// TIA Portal project "Sistema_de_silos" (V16)

(* hardware
DEVICE "S7-1200 station_1"  S7-1200 Station
   slot 0: "Rack_0"  S7-1200 Rack  Rack  V1.0
   slot 1: "PLC_1"  CPU 1215C DC/DC/Rly  6ES7 215-1HG40-0XB0  V4.4
*)

// ===== PLC "PLC_1"  CPU 1215C DC/DC/Rly =====

VAR_GLOBAL   // PLC tag table "Inputs"
   "bt0" AT %I0.0 : Bool;   // botao automático
   "bt1" AT %I0.1 : Bool;   // botao manual
   "bt2" AT %I0.2 : Bool;   // botao reset
   "bt3" AT %I0.3 : Bool;   // botao Emg
   "b01" AT %I0.4 : Bool;   // sensor B01 Silo 1 Nivel Minimo
   "b02" AT %I0.5 : Bool;   // sensor B02 Silo 1 Nivel Maximo
   "b03" AT %I0.6 : Bool;   // sensor B03 Damper aberto silo 2
   "b04" AT %I0.7 : Bool;   // sensor B04 Damper aberto silo 3
   "b05" AT %I1.0 : Bool;   // sensor B05 Silo 2 Nivel Minimo
   "b06" AT %I1.1 : Bool;   // sensor B06 Silo 2 Nivel Máximo
   "b07" AT %I1.2 : Bool;   // sensor B07 Silo 3 Nivel Minimo
   "b08" AT %I1.3 : Bool;   // sensor B08 Silo 3 Nivel Máximo
   "b09" AT %I1.4 : Bool;   // sensor B09 Damper Fechado
   "Reserva" AT %I1.5 : Bool;   // sensor B10 Valvula Silo 2 Fechada
END_VAR

VAR_GLOBAL   // PLC tag table "Outputs"
   "x0.0" AT %Q0.0 : Bool;   // sinalizacao verde
   "x0.1" AT %Q0.1 : Bool;   // sinalizacao amarelo
   "x0.2" AT %Q0.2 : Bool;   // sinalizacao vermelho
   "k0.3" AT %Q0.3 : Bool;   // damper silo 2
   "k0.4" AT %Q0.4 : Bool;   // damper fecha
   "k0.5" AT %Q0.5 : Bool;   // Liga Transportador Silo 2
   "k0.6" AT %Q0.6 : Bool;   // Liga Transportador Silo 3
   "k0.7" AT %Q0.7 : Bool;   // Abre Valvula Silo 1
   "k10" AT %Q1.0 : Bool;   // Abre Valvula Silo 2
   "k11" AT %Q1.1 : Bool;   // damper silo 3
END_VAR

VAR_GLOBAL   // PLC tag table "Memories"
   "Memoria_Auxiliar_Erro_Silo" AT %M0.1 : Bool;
   "ST_FALHA" AT %M0.2 : Bool;
END_VAR

DATA_BLOCK "DB_Geral"   // DB1
{ S7_Optimized_Access := 'TRUE' }
VERSION : 0.1
   VAR
      automatico : Bool;   // Estado automatico
      manual : Bool;   // Estado Manual
      Emg : Bool;   // Estado Emergência
      Falha : Struct   // Estado Falha
         Falha_Desabastecimento_Silo2 : Bool;
         Falha_Desabastecimento_Silo3 : Bool;
         Falha_Desabastecimento_SiloPrincipal : Bool;
         Falha_Sensores_Silo2 : Bool;
         Falha_Sensores_Silo3 : Bool;
         Falha_Sensores_SiloPrincipal : Bool;
      END_STRUCT;
      Diametro_Valvula : Real := 0.1;
      Volume_sensor : Int := 3;
      Volume_maximo_minimo : Int := 7;
      Time_Dint_Valvula : DInt;
      Time_Dint_TempoErro : DInt;
      Time_Valvula : Time;
      Time_TempoErro : Time;
      Sequencia : Struct   // Sequencia Operacional
         Acao : Array[0..50] of Bool;
         Passos : Int;
      END_STRUCT;
      "Status Silo Principal" : Struct   // Status do Silo Principal
         Maximo : Bool;
         Minimo : Bool;
         Desabastecido : Bool;
         Posicao_Produto : Int;
      END_STRUCT;
      "Status Silo 2" : Struct   // Status do Silo 2
         Maximo : Bool;
         Minimo : Bool;
         Desabastecido : Bool;
         Posicao_Produto : Int;
      END_STRUCT;
      "Status Silo 3" : Struct   // Status do Silo 3
         Maximo : Bool;
         Minimo : Bool;
         Desabastecido : Bool;
         Posicao_Produto : Bool;
      END_STRUCT;
      "Status Transportador" : Struct   // Status Transportadores
         "Transportador 1" : Bool;
         "Transportador 2" : Bool;
      END_STRUCT;
      "Status Damper" : Struct   // Status do Damper
         Ligado : Bool;
         "Silo 2" : Bool;
         "Silo 3" : Bool;
      END_STRUCT;
      "Status Valvulas" : Struct   // Status das Valvulas
         "Valvula Silo 2" : Bool;
         "Valvula Silo 3" : Bool;
      END_STRUCT;
   END_VAR
BEGIN
   // Sequencia.Acao[20] : Ação 20
   // Sequencia.Acao[30] : Ação 30
   // Sequencia.Acao[31] : Ação 31
   // Sequencia.Acao[21] : Ação 21
   // Sequencia.Acao[22] : Ação 22
   // Sequencia.Acao[40] : Ação 40
   // Sequencia.Acao[41] : Ação 41
   // Sequencia.Acao[10] : Ação 10
   // Sequencia.Acao[11] : Ação 11
END_DATA_BLOCK

DATA_BLOCK "DB_Inputs"   // DB2
{ S7_Optimized_Access := 'TRUE' }
VERSION : 0.1
   VAR
      bt0 : Bool;   // botao automático
      bt1 : Bool;   // botao manual
      bt2 : Bool;   // botao reset
      bt3 : Bool;   // botao Emg
      bt4 : Bool;   // botao Abre Valvula 2
      bt5 : Bool;   // botao Abre Valvula 3
      b01 : Bool;   // sensor B01 Silo 1 Nivel Minimo
      b02 : Bool;   // sensor B02 Silo 1 Nivel Maximo
      b03 : Bool;   // sensor B03 Damper aberto silo 2
      b04 : Bool;   // sensor B04 Damper aberto silo 3
      b05 : Bool;   // sensor B05 Silo 2 Nivel Minimo
      b06 : Bool;   // sensor B06 Silo 2 Nivel Máximo
      b07 : Bool;   // sensor B07 Silo 3 Nivel Minimo
      b08 : Bool;   // sensor B08 Silo 3 Nivel Máximo
      b09 : Bool;   // sensor B09 Damper Fechado
   END_VAR
BEGIN
END_DATA_BLOCK

DATA_BLOCK "DB_Outputs"   // DB3
{ S7_Optimized_Access := 'TRUE' }
VERSION : 0.1
   VAR
      "x0.0" : Bool;   // sinalizacao verde
      "x0.1" : Bool;   // sinalizacao amarelo
      "x0.2" : Bool;   // sinalizacao vermelho
      "k0.3" : Bool;   // damper Abre silo 2
      "k0.4" : Bool;   // damper Abre silo 3
      "k0.5" : Bool;   // Liga Transportador Silo 2
      "k0.6" : Bool;   // Liga Transportador Silo 3
      "k0.7" : Bool;   // Abre Valvula Silo 2
      k10 : Bool;   // Abre Valvula Silo 3
      k11 : Bool;   // Abastece Silo Principal
   END_VAR
BEGIN
END_DATA_BLOCK

// folder: System blocks/Program resources

DATA_BLOCK "IEC_Timer_0_DB_TOF_VALVULA2"   // DB4
{ S7_Optimized_Access := 'TRUE' }
AUTHOR : Simatic
FAMILY : IEC
NAME : IEC_TMR
VERSION : 1.0
// stored: InstanceOfName IEC_TIMER
"IEC_TIMER"
BEGIN
END_DATA_BLOCK

DATA_BLOCK "IEC_Timer_0_DB_TON_TempoErro"   // DB5
{ S7_Optimized_Access := 'TRUE' }
AUTHOR : Simatic
FAMILY : IEC
NAME : IEC_TMR
VERSION : 1.0
// stored: InstanceOfName IEC_TIMER
"IEC_TIMER"
BEGIN
END_DATA_BLOCK

// folder: (top level)

FUNCTION "FC_Geral" : Void   // FC1, LAD
{ S7_Optimized_Access := 'TRUE' }
VERSION : 0.1
   VAR_TEMP   // added for the SCL form of the ladder/FBD networks
      _w1 : Bool;
   END_VAR
BEGIN

REGION Network 1: Estado Emergencia
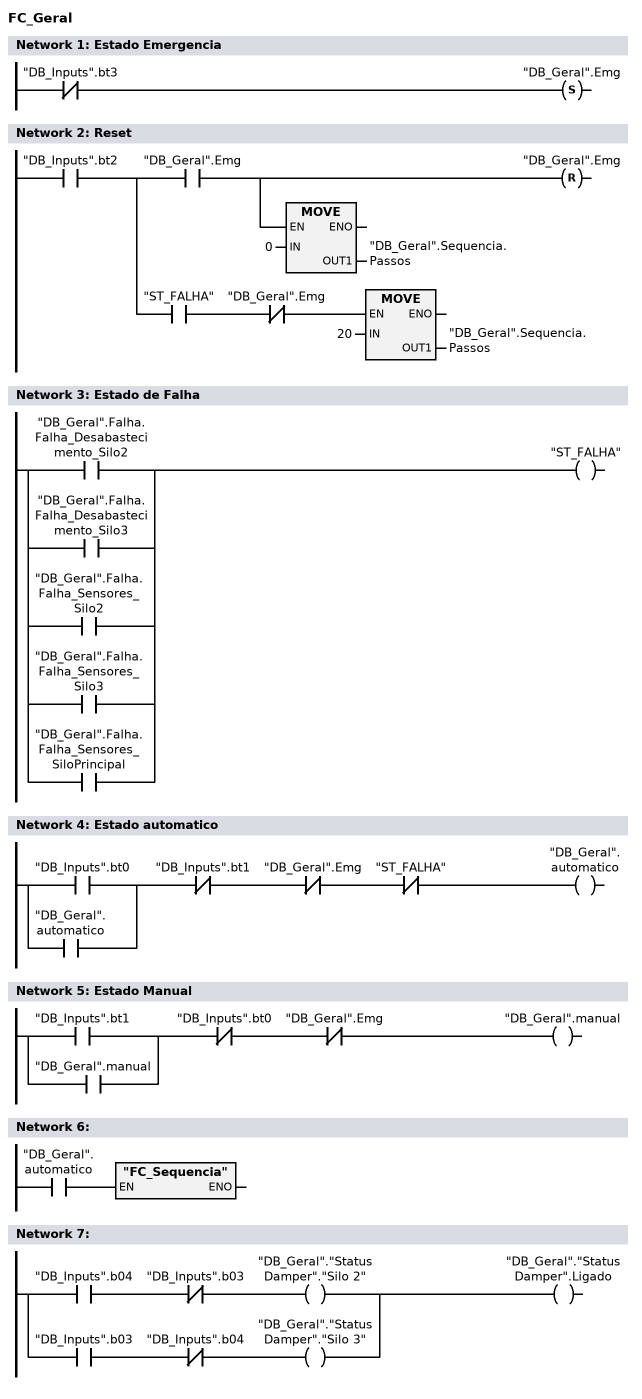
   RUNG wire#powerrail
      I_Contact( "DB_Inputs".bt3 )
      S_Coil( "DB_Geral".Emg )
   END_RUNG
   // the same network as SCL:
   IF NOT "DB_Inputs".bt3 THEN "DB_Geral".Emg := TRUE; END_IF;
END_REGION

REGION Network 2: Reset
   RUNG wire#powerrail
      Contact( "DB_Inputs".bt2 )
      wire#w1
      Contact( "DB_Geral".Emg )
      wire#w2
      R_Coil( "DB_Geral".Emg )
   END_RUNG
   RUNG wire#w2
      Move(in := 0, out1 => "DB_Geral".Sequencia.Passos)
   END_RUNG
   RUNG wire#w1
      Contact( "ST_FALHA" )
      I_Contact( "DB_Geral".Emg )
      Move(in := 20, out1 => "DB_Geral".Sequencia.Passos)
   END_RUNG
   // the same network as SCL:
   #_w1 := "DB_Inputs".bt2 AND "DB_Geral".Emg;
   IF #_w1 THEN
       "DB_Geral".Emg := FALSE;
       "DB_Geral".Sequencia.Passos := 0;
   END_IF;
   IF "DB_Inputs".bt2 AND "ST_FALHA" AND NOT "DB_Geral".Emg THEN "DB_Geral".Sequencia.Passos := 20; END_IF;
END_REGION

REGION Network 3: Estado de Falha
   RUNG wire#powerrail
      Contact( "DB_Geral".Falha.Falha_Desabastecimento_Silo2 )
      wire#w1
      Coil( "ST_FALHA" )
   END_RUNG
   RUNG wire#powerrail
      Contact( "DB_Geral".Falha.Falha_Desabastecimento_Silo3 )
   END_RUNG wire#w1
   RUNG wire#powerrail
      Contact( "DB_Geral".Falha.Falha_Sensores_Silo2 )
   END_RUNG wire#w1
   RUNG wire#powerrail
      Contact( "DB_Geral".Falha.Falha_Sensores_Silo3 )
   END_RUNG wire#w1
   RUNG wire#powerrail
      Contact( "DB_Geral".Falha.Falha_Sensores_SiloPrincipal )
   END_RUNG wire#w1
   // the same network as SCL:
   "ST_FALHA" := "DB_Geral".Falha.Falha_Desabastecimento_Silo2 OR "DB_Geral".Falha.Falha_Desabastecimento_Silo3 OR "DB_Geral".Falha.Falha_Sensores_Silo2 OR "DB_Geral".Falha.Falha_Sensores_Silo3 OR "DB_Geral".Falha.Falha_Sensores_SiloPrincipal;
END_REGION

REGION Network 4: Estado automatico
   RUNG wire#powerrail
      Contact( "DB_Inputs".bt0 )
      wire#w1
      I_Contact( "DB_Inputs".bt1 )
      I_Contact( "DB_Geral".Emg )
      I_Contact( "ST_FALHA" )
      Coil( "DB_Geral".automatico )
   END_RUNG
   RUNG wire#powerrail
      Contact( "DB_Geral".automatico )
   END_RUNG wire#w1
   // the same network as SCL:
   "DB_Geral".automatico := ("DB_Inputs".bt0 OR "DB_Geral".automatico) AND NOT "DB_Inputs".bt1 AND NOT "DB_Geral".Emg AND NOT "ST_FALHA";
END_REGION

REGION Network 5: Estado Manual
   RUNG wire#powerrail
      Contact( "DB_Inputs".bt1 )
      wire#w1
      I_Contact( "DB_Inputs".bt0 )
      I_Contact( "DB_Geral".Emg )
      Coil( "DB_Geral".manual )
   END_RUNG
   RUNG wire#powerrail
      Contact( "DB_Geral".manual )
   END_RUNG wire#w1
   // the same network as SCL:
   "DB_Geral".manual := ("DB_Inputs".bt1 OR "DB_Geral".manual) AND NOT "DB_Inputs".bt0 AND NOT "DB_Geral".Emg;
END_REGION

REGION Network 6
   RUNG wire#powerrail
      Contact( "DB_Geral".automatico )
      "FC_Sequencia"()
   END_RUNG
   // the same network as SCL:
   IF "DB_Geral".automatico THEN "FC_Sequencia"(); END_IF;
END_REGION

REGION Network 7
   RUNG wire#powerrail
      Contact( "DB_Inputs".b04 )
      I_Contact( "DB_Inputs".b03 )
      Coil( "DB_Geral"."Status Damper"."Silo 2" )
      wire#w1
      Coil( "DB_Geral"."Status Damper".Ligado )
   END_RUNG
   RUNG wire#powerrail
      Contact( "DB_Inputs".b03 )
      I_Contact( "DB_Inputs".b04 )
      Coil( "DB_Geral"."Status Damper"."Silo 3" )
   END_RUNG wire#w1
   // the same network as SCL:
   "DB_Geral"."Status Damper"."Silo 2" := "DB_Inputs".b04 AND NOT "DB_Inputs".b03;
   "DB_Geral"."Status Damper"."Silo 3" := "DB_Inputs".b03 AND NOT "DB_Inputs".b04;
   "DB_Geral"."Status Damper".Ligado := "DB_Geral"."Status Damper"."Silo 2" OR "DB_Geral"."Status Damper"."Silo 3";
END_REGION
END_FUNCTION

FUNCTION "FC_Espelho_Outputs" : Void   // FC2, LAD
{ S7_Optimized_Access := 'TRUE' }
VERSION : 0.1
BEGIN

REGION Network 1: sinalizacao verde
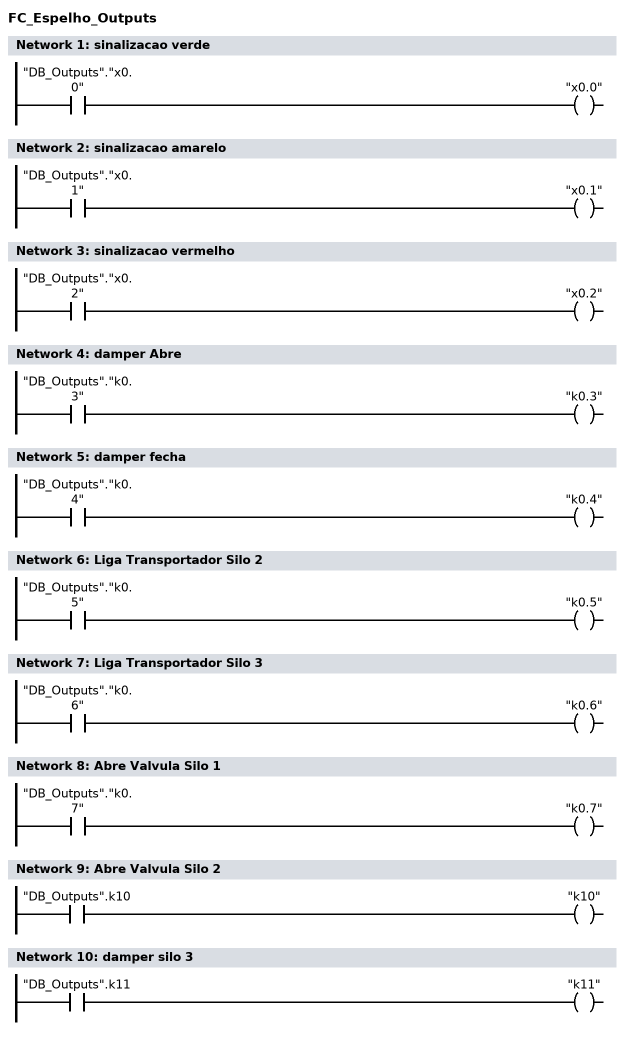
   RUNG wire#powerrail
      Contact( "DB_Outputs"."x0.0" )
      Coil( "x0.0" )
   END_RUNG
   // the same network as SCL:
   "x0.0" := "DB_Outputs"."x0.0";
END_REGION

REGION Network 2: sinalizacao amarelo
   RUNG wire#powerrail
      Contact( "DB_Outputs"."x0.1" )
      Coil( "x0.1" )
   END_RUNG
   // the same network as SCL:
   "x0.1" := "DB_Outputs"."x0.1";
END_REGION

REGION Network 3: sinalizacao vermelho
   RUNG wire#powerrail
      Contact( "DB_Outputs"."x0.2" )
      Coil( "x0.2" )
   END_RUNG
   // the same network as SCL:
   "x0.2" := "DB_Outputs"."x0.2";
END_REGION

REGION Network 4: damper Abre
   RUNG wire#powerrail
      Contact( "DB_Outputs"."k0.3" )
      Coil( "k0.3" )
   END_RUNG
   // the same network as SCL:
   "k0.3" := "DB_Outputs"."k0.3";
END_REGION

REGION Network 5: damper fecha
   RUNG wire#powerrail
      Contact( "DB_Outputs"."k0.4" )
      Coil( "k0.4" )
   END_RUNG
   // the same network as SCL:
   "k0.4" := "DB_Outputs"."k0.4";
END_REGION

REGION Network 6: Liga Transportador Silo 2
   RUNG wire#powerrail
      Contact( "DB_Outputs"."k0.5" )
      Coil( "k0.5" )
   END_RUNG
   // the same network as SCL:
   "k0.5" := "DB_Outputs"."k0.5";
END_REGION

REGION Network 7: Liga Transportador Silo 3
   RUNG wire#powerrail
      Contact( "DB_Outputs"."k0.6" )
      Coil( "k0.6" )
   END_RUNG
   // the same network as SCL:
   "k0.6" := "DB_Outputs"."k0.6";
END_REGION

REGION Network 8: Abre Valvula Silo 1
   RUNG wire#powerrail
      Contact( "DB_Outputs"."k0.7" )
      Coil( "k0.7" )
   END_RUNG
   // the same network as SCL:
   "k0.7" := "DB_Outputs"."k0.7";
END_REGION

REGION Network 9: Abre Valvula Silo 2
   RUNG wire#powerrail
      Contact( "DB_Outputs".k10 )
      Coil( "k10" )
   END_RUNG
   // the same network as SCL:
   "k10" := "DB_Outputs".k10;
END_REGION

REGION Network 10: damper silo 3
   RUNG wire#powerrail
      Contact( "DB_Outputs".k11 )
      Coil( "k11" )
   END_RUNG
   // the same network as SCL:
   "k11" := "DB_Outputs".k11;
END_REGION
END_FUNCTION

FUNCTION "FC_Espelho_Inputs" : Void   // FC3, LAD
{ S7_Optimized_Access := 'TRUE' }
VERSION : 0.1
BEGIN

REGION Network 1: botao automático
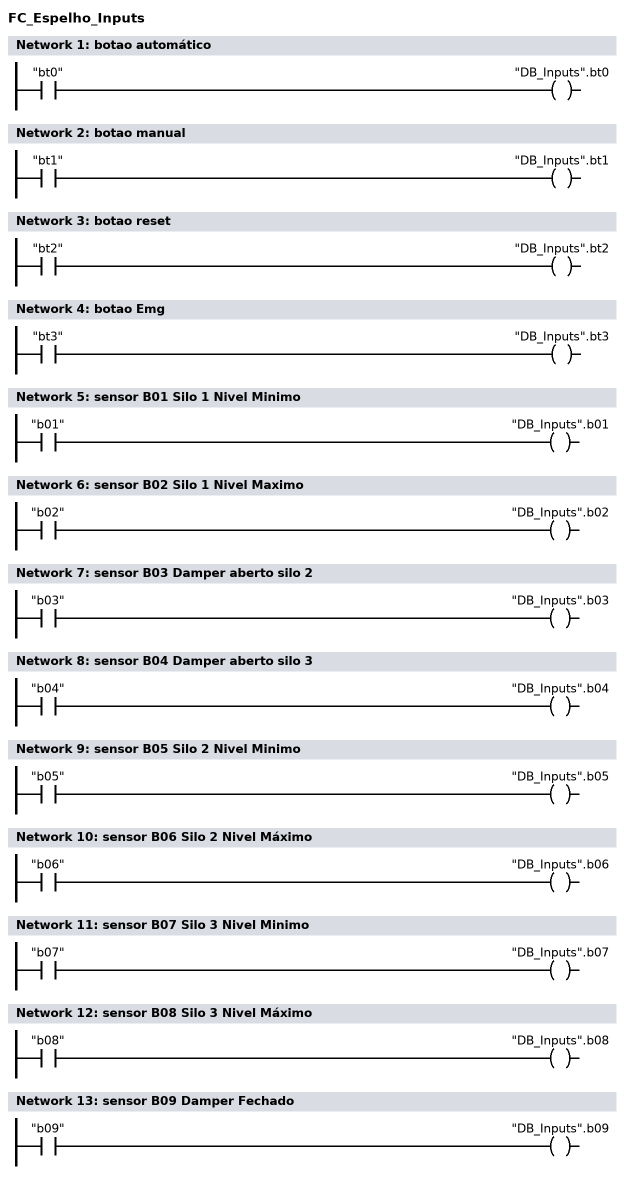
   RUNG wire#powerrail
      Contact( "bt0" )
      Coil( "DB_Inputs".bt0 )
   END_RUNG
   // the same network as SCL:
   "DB_Inputs".bt0 := "bt0";
END_REGION

REGION Network 2: botao manual
   RUNG wire#powerrail
      Contact( "bt1" )
      Coil( "DB_Inputs".bt1 )
   END_RUNG
   // the same network as SCL:
   "DB_Inputs".bt1 := "bt1";
END_REGION

REGION Network 3: botao reset
   RUNG wire#powerrail
      Contact( "bt2" )
      Coil( "DB_Inputs".bt2 )
   END_RUNG
   // the same network as SCL:
   "DB_Inputs".bt2 := "bt2";
END_REGION

REGION Network 4: botao Emg
   RUNG wire#powerrail
      Contact( "bt3" )
      Coil( "DB_Inputs".bt3 )
   END_RUNG
   // the same network as SCL:
   "DB_Inputs".bt3 := "bt3";
END_REGION

REGION Network 5: sensor B01 Silo 1 Nivel Minimo
   RUNG wire#powerrail
      Contact( "b01" )
      Coil( "DB_Inputs".b01 )
   END_RUNG
   // the same network as SCL:
   "DB_Inputs".b01 := "b01";
END_REGION

REGION Network 6: sensor B02 Silo 1 Nivel Maximo
   RUNG wire#powerrail
      Contact( "b02" )
      Coil( "DB_Inputs".b02 )
   END_RUNG
   // the same network as SCL:
   "DB_Inputs".b02 := "b02";
END_REGION

REGION Network 7: sensor B03 Damper aberto silo 2
   RUNG wire#powerrail
      Contact( "b03" )
      Coil( "DB_Inputs".b03 )
   END_RUNG
   // the same network as SCL:
   "DB_Inputs".b03 := "b03";
END_REGION

REGION Network 8: sensor B04 Damper aberto silo 3
   RUNG wire#powerrail
      Contact( "b04" )
      Coil( "DB_Inputs".b04 )
   END_RUNG
   // the same network as SCL:
   "DB_Inputs".b04 := "b04";
END_REGION

REGION Network 9: sensor B05 Silo 2 Nivel Minimo
   RUNG wire#powerrail
      Contact( "b05" )
      Coil( "DB_Inputs".b05 )
   END_RUNG
   // the same network as SCL:
   "DB_Inputs".b05 := "b05";
END_REGION

REGION Network 10: sensor B06 Silo 2 Nivel Máximo
   RUNG wire#powerrail
      Contact( "b06" )
      Coil( "DB_Inputs".b06 )
   END_RUNG
   // the same network as SCL:
   "DB_Inputs".b06 := "b06";
END_REGION

REGION Network 11: sensor B07 Silo 3 Nivel Minimo
   RUNG wire#powerrail
      Contact( "b07" )
      Coil( "DB_Inputs".b07 )
   END_RUNG
   // the same network as SCL:
   "DB_Inputs".b07 := "b07";
END_REGION

REGION Network 12: sensor B08 Silo 3 Nivel Máximo
   RUNG wire#powerrail
      Contact( "b08" )
      Coil( "DB_Inputs".b08 )
   END_RUNG
   // the same network as SCL:
   "DB_Inputs".b08 := "b08";
END_REGION

REGION Network 13: sensor B09 Damper Fechado
   RUNG wire#powerrail
      Contact( "b09" )
      Coil( "DB_Inputs".b09 )
   END_RUNG
   // the same network as SCL:
   "DB_Inputs".b09 := "b09";
END_REGION
END_FUNCTION

FUNCTION "FC_Sequencia" : Void   // FC4, LAD
{ S7_Optimized_Access := 'TRUE' }
VERSION : 0.1
   VAR_TEMP   // added for the SCL form of the ladder/FBD networks
      _w1 : Bool;
   END_VAR
BEGIN

REGION Network 1
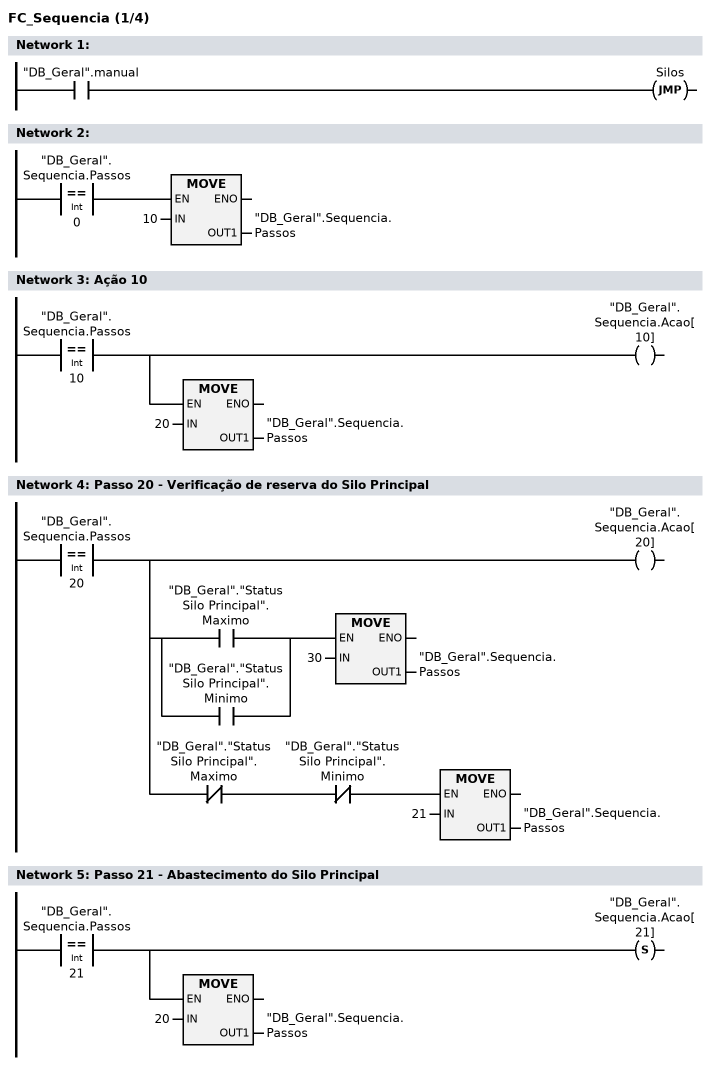
   RUNG wire#powerrail
      Contact( "DB_Geral".manual )
      JumpCoil( Silos )
   END_RUNG
   // the same network as SCL:
   IF "DB_Geral".manual THEN GOTO Silos; END_IF;
END_REGION

REGION Network 2
   RUNG wire#powerrail
      { S7_Templates := "SrcType := Int" } EQ_Contact(in1 := "DB_Geral".Sequencia.Passos, in2 := 0)
      Move(in := 10, out1 => "DB_Geral".Sequencia.Passos)
   END_RUNG
   // the same network as SCL:
   IF "DB_Geral".Sequencia.Passos = 0 THEN "DB_Geral".Sequencia.Passos := 10; END_IF;
END_REGION

REGION Network 3: Ação 10
   RUNG wire#powerrail
      { S7_Templates := "SrcType := Int" } EQ_Contact(in1 := "DB_Geral".Sequencia.Passos, in2 := 10)
      wire#w1
      Coil( "DB_Geral".Sequencia.Acao[10] )
   END_RUNG
   RUNG wire#w1
      Move(in := 20, out1 => "DB_Geral".Sequencia.Passos)
   END_RUNG
   // the same network as SCL:
   "DB_Geral".Sequencia.Acao[10] := "DB_Geral".Sequencia.Passos = 10;
   IF "DB_Geral".Sequencia.Passos = 10 THEN "DB_Geral".Sequencia.Passos := 20; END_IF;
END_REGION

REGION Network 4: Passo 20 - Verificação de reserva do Silo Principal
   RUNG wire#powerrail
      { S7_Templates := "SrcType := Int" } EQ_Contact(in1 := "DB_Geral".Sequencia.Passos, in2 := 20)
      wire#w1
      Coil( "DB_Geral".Sequencia.Acao[20] )
   END_RUNG
   RUNG wire#w1
      Contact( "DB_Geral"."Status Silo Principal".Maximo )
      wire#w2
      Move(in := 30, out1 => "DB_Geral".Sequencia.Passos)
   END_RUNG
   RUNG wire#w1
      Contact( "DB_Geral"."Status Silo Principal".Minimo )
   END_RUNG wire#w2
   RUNG wire#w1
      I_Contact( "DB_Geral"."Status Silo Principal".Maximo )
      I_Contact( "DB_Geral"."Status Silo Principal".Minimo )
      Move(in := 21, out1 => "DB_Geral".Sequencia.Passos)
   END_RUNG
   // the same network as SCL:
   "DB_Geral".Sequencia.Acao[20] := "DB_Geral".Sequencia.Passos = 20;
   #_w1 := "DB_Geral".Sequencia.Passos = 20;
   IF ("DB_Geral".Sequencia.Passos = 20) AND ("DB_Geral"."Status Silo Principal".Maximo OR "DB_Geral"."Status Silo Principal".Minimo) THEN
       "DB_Geral".Sequencia.Passos := 30;
   END_IF;
   IF #_w1 AND NOT "DB_Geral"."Status Silo Principal".Maximo AND NOT "DB_Geral"."Status Silo Principal".Minimo THEN
       "DB_Geral".Sequencia.Passos := 21;
   END_IF;
END_REGION

REGION Network 5: Passo 21 - Abastecimento do Silo Principal
   RUNG wire#powerrail
      { S7_Templates := "SrcType := Int" } EQ_Contact(in1 := "DB_Geral".Sequencia.Passos, in2 := 21)
      wire#w1
      S_Coil( "DB_Geral".Sequencia.Acao[21] )
   END_RUNG
   RUNG wire#w1
      Move(in := 20, out1 => "DB_Geral".Sequencia.Passos)
   END_RUNG
   // the same network as SCL:
   IF "DB_Geral".Sequencia.Passos = 21 THEN
       "DB_Geral".Sequencia.Acao[21] := TRUE;
       "DB_Geral".Sequencia.Passos := 20;
   END_IF;
END_REGION

REGION Network 6: Passo 30 - Verificação do Silo 2
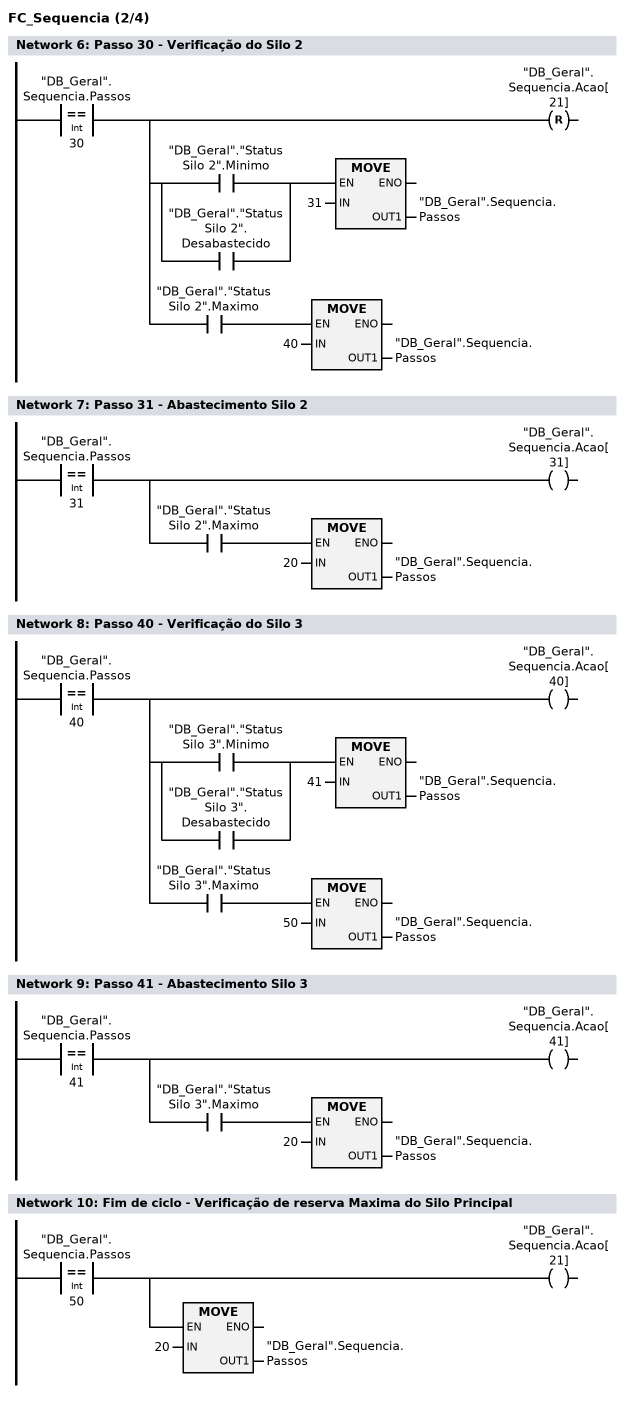
   RUNG wire#powerrail
      { S7_Templates := "SrcType := Int" } EQ_Contact(in1 := "DB_Geral".Sequencia.Passos, in2 := 30)
      wire#w1
      R_Coil( "DB_Geral".Sequencia.Acao[21] )
   END_RUNG
   RUNG wire#w1
      Contact( "DB_Geral"."Status Silo 2".Minimo )
      wire#w2
      Move(in := 31, out1 => "DB_Geral".Sequencia.Passos)
   END_RUNG
   RUNG wire#w1
      Contact( "DB_Geral"."Status Silo 2".Desabastecido )
   END_RUNG wire#w2
   RUNG wire#w1
      Contact( "DB_Geral"."Status Silo 2".Maximo )
      Move(in := 40, out1 => "DB_Geral".Sequencia.Passos)
   END_RUNG
   // the same network as SCL:
   #_w1 := "DB_Geral".Sequencia.Passos = 30;
   IF #_w1 THEN "DB_Geral".Sequencia.Acao[21] := FALSE; END_IF;
   IF #_w1 AND ("DB_Geral"."Status Silo 2".Minimo OR "DB_Geral"."Status Silo 2".Desabastecido) THEN
       "DB_Geral".Sequencia.Passos := 31;
   END_IF;
   IF #_w1 AND "DB_Geral"."Status Silo 2".Maximo THEN "DB_Geral".Sequencia.Passos := 40; END_IF;
END_REGION

REGION Network 7: Passo 31 - Abastecimento Silo 2
   RUNG wire#powerrail
      { S7_Templates := "SrcType := Int" } EQ_Contact(in1 := "DB_Geral".Sequencia.Passos, in2 := 31)
      wire#w1
      Coil( "DB_Geral".Sequencia.Acao[31] )
   END_RUNG
   RUNG wire#w1
      Contact( "DB_Geral"."Status Silo 2".Maximo )
      Move(in := 20, out1 => "DB_Geral".Sequencia.Passos)
   END_RUNG
   // the same network as SCL:
   "DB_Geral".Sequencia.Acao[31] := "DB_Geral".Sequencia.Passos = 31;
   IF ("DB_Geral".Sequencia.Passos = 31) AND "DB_Geral"."Status Silo 2".Maximo THEN
       "DB_Geral".Sequencia.Passos := 20;
   END_IF;
END_REGION

REGION Network 8: Passo 40 - Verificação do Silo 3
   RUNG wire#powerrail
      { S7_Templates := "SrcType := Int" } EQ_Contact(in1 := "DB_Geral".Sequencia.Passos, in2 := 40)
      wire#w1
      Coil( "DB_Geral".Sequencia.Acao[40] )
   END_RUNG
   RUNG wire#w1
      Contact( "DB_Geral"."Status Silo 3".Minimo )
      wire#w2
      Move(in := 41, out1 => "DB_Geral".Sequencia.Passos)
   END_RUNG
   RUNG wire#w1
      Contact( "DB_Geral"."Status Silo 3".Desabastecido )
   END_RUNG wire#w2
   RUNG wire#w1
      Contact( "DB_Geral"."Status Silo 3".Maximo )
      Move(in := 50, out1 => "DB_Geral".Sequencia.Passos)
   END_RUNG
   // the same network as SCL:
   "DB_Geral".Sequencia.Acao[40] := "DB_Geral".Sequencia.Passos = 40;
   #_w1 := "DB_Geral".Sequencia.Passos = 40;
   IF ("DB_Geral".Sequencia.Passos = 40) AND ("DB_Geral"."Status Silo 3".Minimo OR "DB_Geral"."Status Silo 3".Desabastecido) THEN
       "DB_Geral".Sequencia.Passos := 41;
   END_IF;
   IF #_w1 AND "DB_Geral"."Status Silo 3".Maximo THEN "DB_Geral".Sequencia.Passos := 50; END_IF;
END_REGION

REGION Network 9: Passo 41 - Abastecimento Silo 3
   RUNG wire#powerrail
      { S7_Templates := "SrcType := Int" } EQ_Contact(in1 := "DB_Geral".Sequencia.Passos, in2 := 41)
      wire#w1
      Coil( "DB_Geral".Sequencia.Acao[41] )
   END_RUNG
   RUNG wire#w1
      Contact( "DB_Geral"."Status Silo 3".Maximo )
      Move(in := 20, out1 => "DB_Geral".Sequencia.Passos)
   END_RUNG
   // the same network as SCL:
   "DB_Geral".Sequencia.Acao[41] := "DB_Geral".Sequencia.Passos = 41;
   IF ("DB_Geral".Sequencia.Passos = 41) AND "DB_Geral"."Status Silo 3".Maximo THEN
       "DB_Geral".Sequencia.Passos := 20;
   END_IF;
END_REGION

REGION Network 10: Fim de ciclo - Verificação de reserva Maxima do Silo Principal
   RUNG wire#powerrail
      { S7_Templates := "SrcType := Int" } EQ_Contact(in1 := "DB_Geral".Sequencia.Passos, in2 := 50)
      wire#w1
      Coil( "DB_Geral".Sequencia.Acao[21] )
   END_RUNG
   RUNG wire#w1
      Move(in := 20, out1 => "DB_Geral".Sequencia.Passos)
   END_RUNG
   // the same network as SCL:
   "DB_Geral".Sequencia.Acao[21] := "DB_Geral".Sequencia.Passos = 50;
   IF "DB_Geral".Sequencia.Passos = 50 THEN "DB_Geral".Sequencia.Passos := 20; END_IF;
END_REGION

REGION Network 11
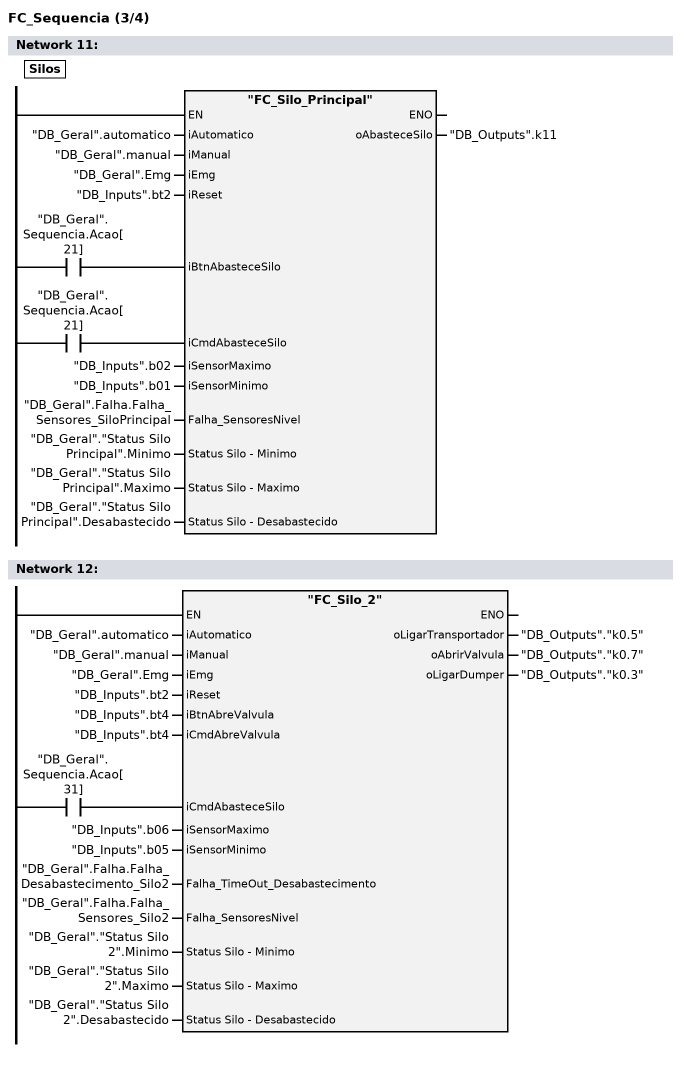
   Label( Silos )
   RUNG wire#powerrail
      "FC_Silo_Principal"(iBtnAbasteceSilo := wire#w1, iCmdAbasteceSilo := wire#w2, iAutomatico := "DB_Geral".automatico, iManual := "DB_Geral".manual, iEmg := "DB_Geral".Emg, iReset := "DB_Inputs".bt2, iSensorMaximo := "DB_Inputs".b02, iSensorMinimo := "DB_Inputs".b01, Falha_SensoresNivel := "DB_Geral".Falha.Falha_Sensores_SiloPrincipal, "Status Silo - Minimo" := "DB_Geral"."Status Silo Principal".Minimo, "Status Silo - Maximo" := "DB_Geral"."Status Silo Principal".Maximo, "Status Silo - Desabastecido" := "DB_Geral"."Status Silo Principal".Desabastecido, oAbasteceSilo => "DB_Outputs".k11)
   END_RUNG
   RUNG wire#powerrail
      Contact( "DB_Geral".Sequencia.Acao[21] )
   END_RUNG wire#w1
   RUNG wire#powerrail
      Contact( "DB_Geral".Sequencia.Acao[21] )
   END_RUNG wire#w2
   // the same network as SCL:
   Silos:
   "FC_Silo_Principal"(iAutomatico := "DB_Geral".automatico,
                       iManual := "DB_Geral".manual,
                       iEmg := "DB_Geral".Emg,
                       iReset := "DB_Inputs".bt2,
                       iBtnAbasteceSilo := "DB_Geral".Sequencia.Acao[21],
                       iCmdAbasteceSilo := "DB_Geral".Sequencia.Acao[21],
                       iSensorMaximo := "DB_Inputs".b02,
                       iSensorMinimo := "DB_Inputs".b01,
                       Falha_SensoresNivel := "DB_Geral".Falha.Falha_Sensores_SiloPrincipal,
                       "Status Silo - Minimo" := "DB_Geral"."Status Silo Principal".Minimo,
                       "Status Silo - Maximo" := "DB_Geral"."Status Silo Principal".Maximo,
                       "Status Silo - Desabastecido" := "DB_Geral"."Status Silo Principal".Desabastecido,
                       oAbasteceSilo => "DB_Outputs".k11);
END_REGION

REGION Network 12
   RUNG wire#powerrail
      "FC_Silo_2"(iCmdAbasteceSilo := wire#w1, iAutomatico := "DB_Geral".automatico, iManual := "DB_Geral".manual, iEmg := "DB_Geral".Emg, iReset := "DB_Inputs".bt2, iBtnAbreValvula := "DB_Inputs".bt4, iCmdAbreValvula := "DB_Inputs".bt4, iSensorMaximo := "DB_Inputs".b06, iSensorMinimo := "DB_Inputs".b05, Falha_TimeOut_Desabastecimento := "DB_Geral".Falha.Falha_Desabastecimento_Silo2, Falha_SensoresNivel := "DB_Geral".Falha.Falha_Sensores_Silo2, "Status Silo - Minimo" := "DB_Geral"."Status Silo 2".Minimo, "Status Silo - Maximo" := "DB_Geral"."Status Silo 2".Maximo, "Status Silo - Desabastecido" := "DB_Geral"."Status Silo 2".Desabastecido, oLigarTransportador => "DB_Outputs"."k0.5", oAbrirValvula => "DB_Outputs"."k0.7", oLigarDumper => "DB_Outputs"."k0.3")
   END_RUNG
   RUNG wire#powerrail
      Contact( "DB_Geral".Sequencia.Acao[31] )
   END_RUNG wire#w1
   // the same network as SCL:
   "FC_Silo_2"(iAutomatico := "DB_Geral".automatico,
               iManual := "DB_Geral".manual,
               iEmg := "DB_Geral".Emg,
               iReset := "DB_Inputs".bt2,
               iBtnAbreValvula := "DB_Inputs".bt4,
               iCmdAbreValvula := "DB_Inputs".bt4,
               iCmdAbasteceSilo := "DB_Geral".Sequencia.Acao[31],
               iSensorMaximo := "DB_Inputs".b06,
               iSensorMinimo := "DB_Inputs".b05,
               Falha_TimeOut_Desabastecimento := "DB_Geral".Falha.Falha_Desabastecimento_Silo2,
               Falha_SensoresNivel := "DB_Geral".Falha.Falha_Sensores_Silo2,
               "Status Silo - Minimo" := "DB_Geral"."Status Silo 2".Minimo,
               "Status Silo - Maximo" := "DB_Geral"."Status Silo 2".Maximo,
               "Status Silo - Desabastecido" := "DB_Geral"."Status Silo 2".Desabastecido,
               oLigarTransportador => "DB_Outputs"."k0.5",
               oAbrirValvula => "DB_Outputs"."k0.7",
               oLigarDumper => "DB_Outputs"."k0.3");
END_REGION

REGION Network 13
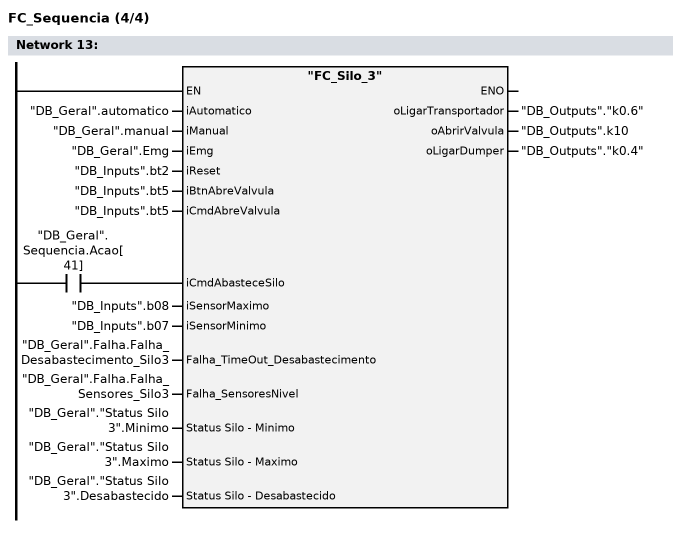
   RUNG wire#powerrail
      "FC_Silo_3"(iCmdAbasteceSilo := wire#w1, iAutomatico := "DB_Geral".automatico, iManual := "DB_Geral".manual, iEmg := "DB_Geral".Emg, iReset := "DB_Inputs".bt2, iBtnAbreValvula := "DB_Inputs".bt5, iCmdAbreValvula := "DB_Inputs".bt5, iSensorMaximo := "DB_Inputs".b08, iSensorMinimo := "DB_Inputs".b07, Falha_TimeOut_Desabastecimento := "DB_Geral".Falha.Falha_Desabastecimento_Silo3, Falha_SensoresNivel := "DB_Geral".Falha.Falha_Sensores_Silo3, "Status Silo - Minimo" := "DB_Geral"."Status Silo 3".Minimo, "Status Silo - Maximo" := "DB_Geral"."Status Silo 3".Maximo, "Status Silo - Desabastecido" := "DB_Geral"."Status Silo 3".Desabastecido, oLigarTransportador => "DB_Outputs"."k0.6", oAbrirValvula => "DB_Outputs".k10, oLigarDumper => "DB_Outputs"."k0.4")
   END_RUNG
   RUNG wire#powerrail
      Contact( "DB_Geral".Sequencia.Acao[41] )
   END_RUNG wire#w1
   // the same network as SCL:
   "FC_Silo_3"(iAutomatico := "DB_Geral".automatico,
               iManual := "DB_Geral".manual,
               iEmg := "DB_Geral".Emg,
               iReset := "DB_Inputs".bt2,
               iBtnAbreValvula := "DB_Inputs".bt5,
               iCmdAbreValvula := "DB_Inputs".bt5,
               iCmdAbasteceSilo := "DB_Geral".Sequencia.Acao[41],
               iSensorMaximo := "DB_Inputs".b08,
               iSensorMinimo := "DB_Inputs".b07,
               Falha_TimeOut_Desabastecimento := "DB_Geral".Falha.Falha_Desabastecimento_Silo3,
               Falha_SensoresNivel := "DB_Geral".Falha.Falha_Sensores_Silo3,
               "Status Silo - Minimo" := "DB_Geral"."Status Silo 3".Minimo,
               "Status Silo - Maximo" := "DB_Geral"."Status Silo 3".Maximo,
               "Status Silo - Desabastecido" := "DB_Geral"."Status Silo 3".Desabastecido,
               oLigarTransportador => "DB_Outputs"."k0.6",
               oAbrirValvula => "DB_Outputs".k10,
               oLigarDumper => "DB_Outputs"."k0.4");
END_REGION
END_FUNCTION

FUNCTION "FC_Silo_2" : Void   // FC5, LAD
{ S7_Optimized_Access := 'TRUE' }
VERSION : 0.1
   VAR_INPUT
      iAutomatico : Bool;
      iManual : Bool;
      iEmg : Bool;
      iReset : Bool;
      iBtnAbreValvula : Bool;
      iCmdAbreValvula : Bool;
      iCmdAbasteceSilo : Bool;
      iSensorMaximo : Bool;
      iSensorMinimo : Bool;
   END_VAR
   VAR_OUTPUT
      oLigarTransportador : Bool;
      oAbrirValvula : Bool;
      oLigarDumper : Bool;
   END_VAR
   VAR_IN_OUT
      Falha_TimeOut_Desabastecimento : Bool;
      Falha_SensoresNivel : Bool;
      "Status Silo - Minimo" : Bool;
      "Status Silo - Maximo" : Bool;
      "Status Silo - Desabastecido" : Bool;
   END_VAR
   VAR CONSTANT
      Velocidade_fluxo : Int := 12;
   END_VAR
BEGIN

REGION Network 1
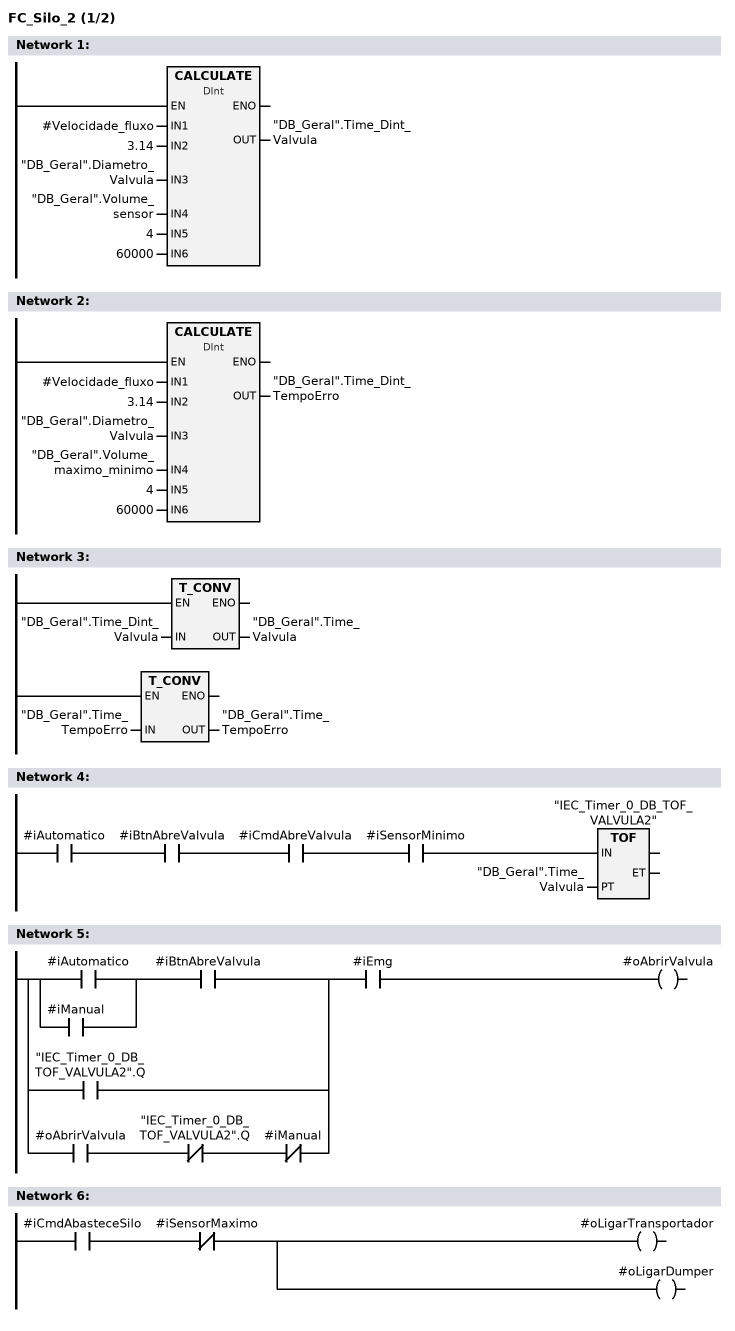
   RUNG wire#powerrail
      { S7_Templates := "SrcType := DInt"; S7_Expression := "(IN4 / (IN1* ((IN2*IN3*IN3) / IN5))) * IN6" } Calculate(in1 := #Velocidade_fluxo, in2 := 3.14, in3 := "DB_Geral".Diametro_Valvula, in4 := "DB_Geral".Volume_sensor, in5 := 4, in6 := 60000, out => "DB_Geral".Time_Dint_Valvula)
   END_RUNG
   // the same network as SCL:
   "DB_Geral".Time_Dint_Valvula := ("DB_Geral".Volume_sensor / (#Velocidade_fluxo* ((3.14*"DB_Geral".Diametro_Valvula*"DB_Geral".Diametro_Valvula) / 4))) * 60000;
END_REGION

REGION Network 2
   RUNG wire#powerrail
      { S7_Templates := "SrcType := DInt"; S7_Expression := "(IN4 / (IN1* ((IN2*IN3*IN3) / IN5))) * IN6" } Calculate(in1 := #Velocidade_fluxo, in2 := 3.14, in3 := "DB_Geral".Diametro_Valvula, in4 := "DB_Geral".Volume_maximo_minimo, in5 := 4, in6 := 60000, out => "DB_Geral".Time_Dint_TempoErro)
   END_RUNG
   // the same network as SCL:
   "DB_Geral".Time_Dint_TempoErro := ("DB_Geral".Volume_maximo_minimo / (#Velocidade_fluxo* ((3.14*"DB_Geral".Diametro_Valvula*"DB_Geral".Diametro_Valvula) / 4))) * 60000;
END_REGION

REGION Network 3
   "DB_Geral".Time_Valvula := T_CONV(IN := "DB_Geral".Time_Dint_Valvula);
   "DB_Geral".Time_TempoErro := T_CONV(IN := "DB_Geral".Time_TempoErro);
END_REGION

REGION Network 4
   "IEC_Timer_0_DB_TOF_VALVULA2".TOF(IN := #iAutomatico AND #iBtnAbreValvula AND #iCmdAbreValvula AND #iSensorMinimo,
                           PT := "DB_Geral".Time_Valvula);
END_REGION

REGION Network 5
   RUNG wire#powerrail
      Contact( #iAutomatico )
      wire#w1
      Contact( #iBtnAbreValvula )
      wire#w2
      Contact( #iEmg )
      Coil( #oAbrirValvula )
   END_RUNG
   RUNG wire#powerrail
      Contact( #iManual )
   END_RUNG wire#w1
   RUNG wire#powerrail
      Contact( "IEC_Timer_0_DB_TOF_VALVULA2".Q )
   END_RUNG wire#w2
   RUNG wire#powerrail
      Contact( #oAbrirValvula )
      I_Contact( "IEC_Timer_0_DB_TOF_VALVULA2".Q )
      I_Contact( #iManual )
   END_RUNG wire#w2
   // the same network as SCL:
   #oAbrirValvula := (((#iAutomatico OR #iManual) AND #iBtnAbreValvula) OR "IEC_Timer_0_DB_TOF_VALVULA2".Q OR (#oAbrirValvula AND NOT "IEC_Timer_0_DB_TOF_VALVULA2".Q AND NOT #iManual)) AND #iEmg;
END_REGION

REGION Network 6
   RUNG wire#powerrail
      Contact( #iCmdAbasteceSilo )
      I_Contact( #iSensorMaximo )
      wire#w1
      Coil( #oLigarTransportador )
   END_RUNG
   RUNG wire#w1
      Coil( #oLigarDumper )
   END_RUNG
   // the same network as SCL:
   #oLigarTransportador := #iCmdAbasteceSilo AND NOT #iSensorMaximo;
   #oLigarDumper := #oLigarTransportador;
END_REGION

REGION Network 7: Silo Principal - Reserva do produto
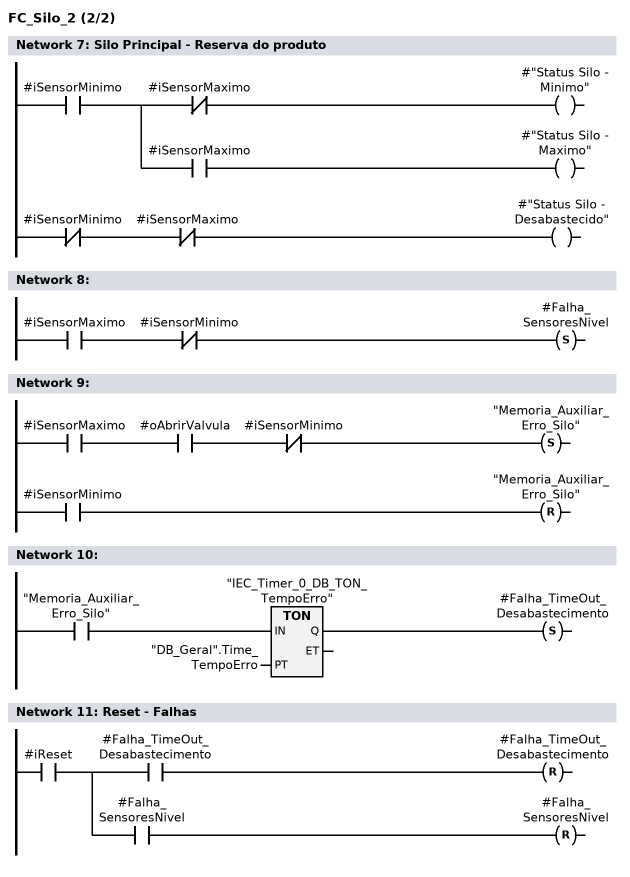
   RUNG wire#powerrail
      Contact( #iSensorMinimo )
      wire#w1
      I_Contact( #iSensorMaximo )
      Coil( #"Status Silo - Minimo" )
   END_RUNG
   RUNG wire#w1
      Contact( #iSensorMaximo )
      Coil( #"Status Silo - Maximo" )
   END_RUNG
   RUNG wire#powerrail
      I_Contact( #iSensorMinimo )
      I_Contact( #iSensorMaximo )
      Coil( #"Status Silo - Desabastecido" )
   END_RUNG
   // the same network as SCL:
   #"Status Silo - Minimo" := #iSensorMinimo AND NOT #iSensorMaximo;
   #"Status Silo - Maximo" := #iSensorMinimo AND #iSensorMaximo;
   #"Status Silo - Desabastecido" := NOT #iSensorMinimo AND NOT #iSensorMaximo;
END_REGION

REGION Network 8
   RUNG wire#powerrail
      Contact( #iSensorMaximo )
      I_Contact( #iSensorMinimo )
      S_Coil( #Falha_SensoresNivel )
   END_RUNG
   // the same network as SCL:
   IF #iSensorMaximo AND NOT #iSensorMinimo THEN #Falha_SensoresNivel := TRUE; END_IF;
END_REGION

REGION Network 9
   RUNG wire#powerrail
      Contact( #iSensorMaximo )
      Contact( #oAbrirValvula )
      I_Contact( #iSensorMinimo )
      S_Coil( "Memoria_Auxiliar_Erro_Silo" )
   END_RUNG
   RUNG wire#powerrail
      Contact( #iSensorMinimo )
      R_Coil( "Memoria_Auxiliar_Erro_Silo" )
   END_RUNG
   // the same network as SCL:
   IF #iSensorMaximo AND #oAbrirValvula AND NOT #iSensorMinimo THEN
       "Memoria_Auxiliar_Erro_Silo" := TRUE;
   END_IF;
   IF #iSensorMinimo THEN "Memoria_Auxiliar_Erro_Silo" := FALSE; END_IF;
END_REGION

REGION Network 10
   "IEC_Timer_0_DB_TON_TempoErro".TON(IN := "Memoria_Auxiliar_Erro_Silo", PT := "DB_Geral".Time_TempoErro);
   IF "IEC_Timer_0_DB_TON_TempoErro".Q THEN #Falha_TimeOut_Desabastecimento := TRUE; END_IF;
END_REGION

REGION Network 11: Reset - Falhas
   RUNG wire#powerrail
      Contact( #iReset )
      wire#w1
      Contact( #Falha_TimeOut_Desabastecimento )
      R_Coil( #Falha_TimeOut_Desabastecimento )
   END_RUNG
   RUNG wire#w1
      Contact( #Falha_SensoresNivel )
      R_Coil( #Falha_SensoresNivel )
   END_RUNG
   // the same network as SCL:
   IF #iReset AND #Falha_TimeOut_Desabastecimento THEN #Falha_TimeOut_Desabastecimento := FALSE; END_IF;
   IF #iReset AND #Falha_SensoresNivel THEN #Falha_SensoresNivel := FALSE; END_IF;
END_REGION
END_FUNCTION

FUNCTION "FC_Silo_3" : Void   // FC5, LAD
{ S7_Optimized_Access := 'TRUE' }
VERSION : 0.1
   VAR_INPUT
      iAutomatico : Bool;
      iManual : Bool;
      iEmg : Bool;
      iReset : Bool;
      iBtnAbreValvula : Bool;
      iCmdAbreValvula : Bool;
      iCmdAbasteceSilo : Bool;
      iSensorMaximo : Bool;
      iSensorMinimo : Bool;
   END_VAR
   VAR_OUTPUT
      oLigarTransportador : Bool;
      oAbrirValvula : Bool;
      oLigarDumper : Bool;
   END_VAR
   VAR_IN_OUT
      Falha_TimeOut_Desabastecimento : Bool;
      Falha_SensoresNivel : Bool;
      "Status Silo - Minimo" : Bool;
      "Status Silo - Maximo" : Bool;
      "Status Silo - Desabastecido" : Bool;
   END_VAR
   VAR CONSTANT
      Velocidade_fluxo : Int := 12;
   END_VAR
BEGIN

REGION Network 1
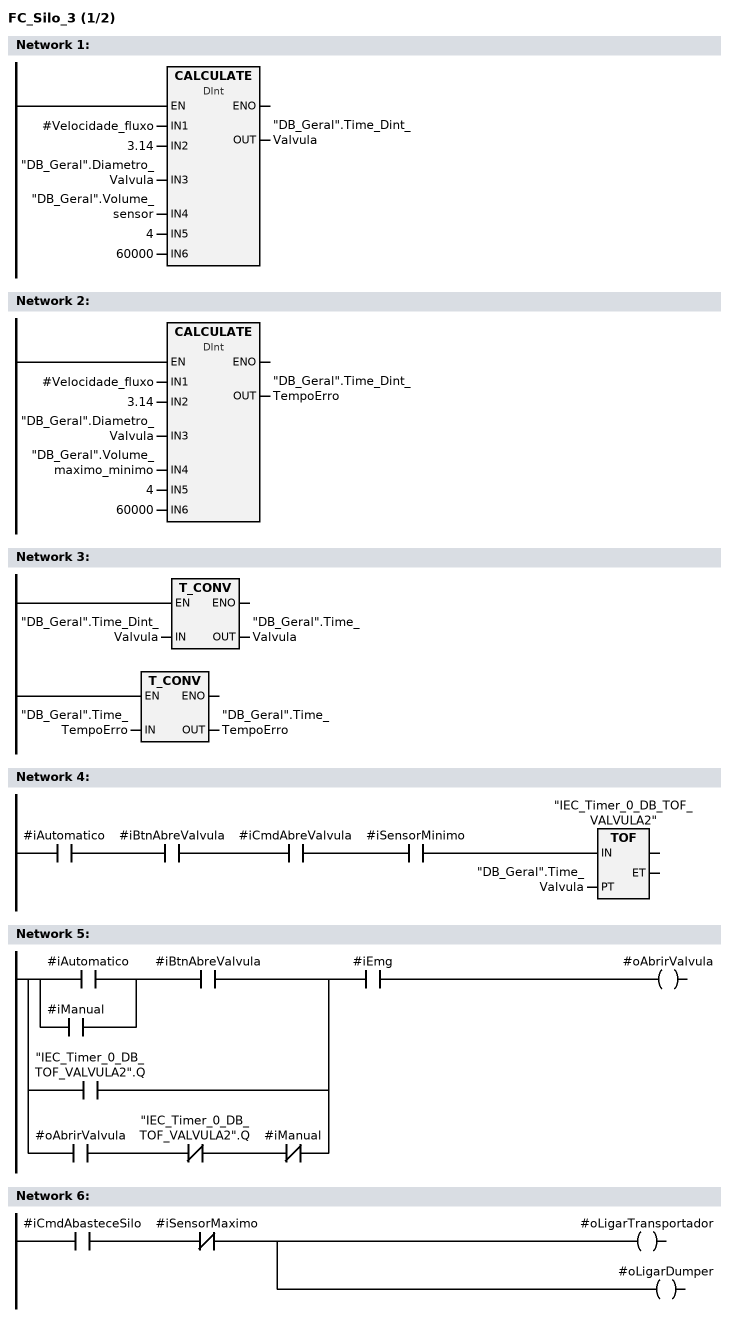
   RUNG wire#powerrail
      { S7_Templates := "SrcType := DInt"; S7_Expression := "(IN4 / (IN1* ((IN2*IN3*IN3) / IN5))) * IN6" } Calculate(in1 := #Velocidade_fluxo, in2 := 3.14, in3 := "DB_Geral".Diametro_Valvula, in4 := "DB_Geral".Volume_sensor, in5 := 4, in6 := 60000, out => "DB_Geral".Time_Dint_Valvula)
   END_RUNG
   // the same network as SCL:
   "DB_Geral".Time_Dint_Valvula := ("DB_Geral".Volume_sensor / (#Velocidade_fluxo* ((3.14*"DB_Geral".Diametro_Valvula*"DB_Geral".Diametro_Valvula) / 4))) * 60000;
END_REGION

REGION Network 2
   RUNG wire#powerrail
      { S7_Templates := "SrcType := DInt"; S7_Expression := "(IN4 / (IN1* ((IN2*IN3*IN3) / IN5))) * IN6" } Calculate(in1 := #Velocidade_fluxo, in2 := 3.14, in3 := "DB_Geral".Diametro_Valvula, in4 := "DB_Geral".Volume_maximo_minimo, in5 := 4, in6 := 60000, out => "DB_Geral".Time_Dint_TempoErro)
   END_RUNG
   // the same network as SCL:
   "DB_Geral".Time_Dint_TempoErro := ("DB_Geral".Volume_maximo_minimo / (#Velocidade_fluxo* ((3.14*"DB_Geral".Diametro_Valvula*"DB_Geral".Diametro_Valvula) / 4))) * 60000;
END_REGION

REGION Network 3
   "DB_Geral".Time_Valvula := T_CONV(IN := "DB_Geral".Time_Dint_Valvula);
   "DB_Geral".Time_TempoErro := T_CONV(IN := "DB_Geral".Time_TempoErro);
END_REGION

REGION Network 4
   "IEC_Timer_0_DB_TOF_VALVULA2".TOF(IN := #iAutomatico AND #iBtnAbreValvula AND #iCmdAbreValvula AND #iSensorMinimo,
                           PT := "DB_Geral".Time_Valvula);
END_REGION

REGION Network 5
   RUNG wire#powerrail
      Contact( #iAutomatico )
      wire#w1
      Contact( #iBtnAbreValvula )
      wire#w2
      Contact( #iEmg )
      Coil( #oAbrirValvula )
   END_RUNG
   RUNG wire#powerrail
      Contact( #iManual )
   END_RUNG wire#w1
   RUNG wire#powerrail
      Contact( "IEC_Timer_0_DB_TOF_VALVULA2".Q )
   END_RUNG wire#w2
   RUNG wire#powerrail
      Contact( #oAbrirValvula )
      I_Contact( "IEC_Timer_0_DB_TOF_VALVULA2".Q )
      I_Contact( #iManual )
   END_RUNG wire#w2
   // the same network as SCL:
   #oAbrirValvula := (((#iAutomatico OR #iManual) AND #iBtnAbreValvula) OR "IEC_Timer_0_DB_TOF_VALVULA2".Q OR (#oAbrirValvula AND NOT "IEC_Timer_0_DB_TOF_VALVULA2".Q AND NOT #iManual)) AND #iEmg;
END_REGION

REGION Network 6
   RUNG wire#powerrail
      Contact( #iCmdAbasteceSilo )
      I_Contact( #iSensorMaximo )
      wire#w1
      Coil( #oLigarTransportador )
   END_RUNG
   RUNG wire#w1
      Coil( #oLigarDumper )
   END_RUNG
   // the same network as SCL:
   #oLigarTransportador := #iCmdAbasteceSilo AND NOT #iSensorMaximo;
   #oLigarDumper := #oLigarTransportador;
END_REGION

REGION Network 7: Silo Principal - Reserva do produto
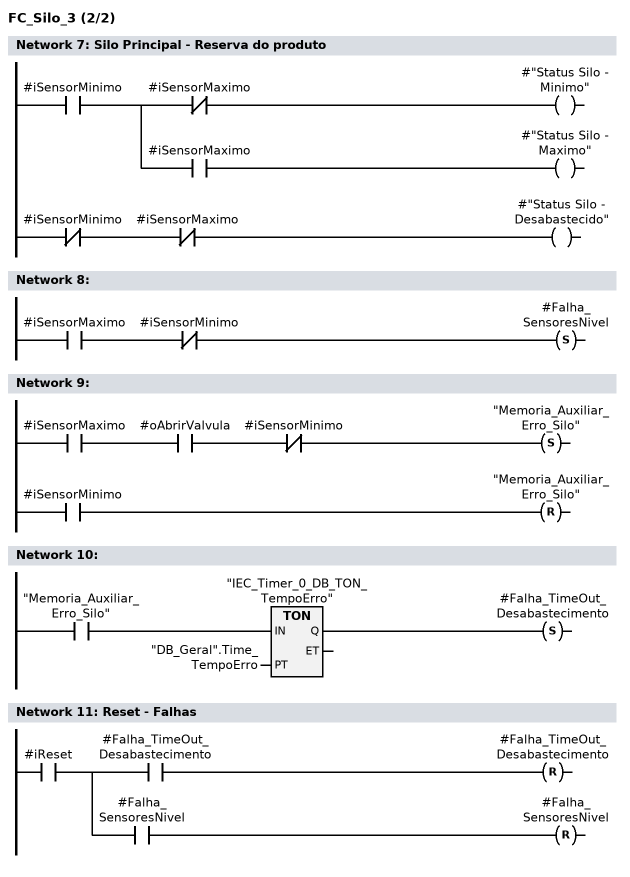
   RUNG wire#powerrail
      Contact( #iSensorMinimo )
      wire#w1
      I_Contact( #iSensorMaximo )
      Coil( #"Status Silo - Minimo" )
   END_RUNG
   RUNG wire#w1
      Contact( #iSensorMaximo )
      Coil( #"Status Silo - Maximo" )
   END_RUNG
   RUNG wire#powerrail
      I_Contact( #iSensorMinimo )
      I_Contact( #iSensorMaximo )
      Coil( #"Status Silo - Desabastecido" )
   END_RUNG
   // the same network as SCL:
   #"Status Silo - Minimo" := #iSensorMinimo AND NOT #iSensorMaximo;
   #"Status Silo - Maximo" := #iSensorMinimo AND #iSensorMaximo;
   #"Status Silo - Desabastecido" := NOT #iSensorMinimo AND NOT #iSensorMaximo;
END_REGION

REGION Network 8
   RUNG wire#powerrail
      Contact( #iSensorMaximo )
      I_Contact( #iSensorMinimo )
      S_Coil( #Falha_SensoresNivel )
   END_RUNG
   // the same network as SCL:
   IF #iSensorMaximo AND NOT #iSensorMinimo THEN #Falha_SensoresNivel := TRUE; END_IF;
END_REGION

REGION Network 9
   RUNG wire#powerrail
      Contact( #iSensorMaximo )
      Contact( #oAbrirValvula )
      I_Contact( #iSensorMinimo )
      S_Coil( "Memoria_Auxiliar_Erro_Silo" )
   END_RUNG
   RUNG wire#powerrail
      Contact( #iSensorMinimo )
      R_Coil( "Memoria_Auxiliar_Erro_Silo" )
   END_RUNG
   // the same network as SCL:
   IF #iSensorMaximo AND #oAbrirValvula AND NOT #iSensorMinimo THEN
       "Memoria_Auxiliar_Erro_Silo" := TRUE;
   END_IF;
   IF #iSensorMinimo THEN "Memoria_Auxiliar_Erro_Silo" := FALSE; END_IF;
END_REGION

REGION Network 10
   "IEC_Timer_0_DB_TON_TempoErro".TON(IN := "Memoria_Auxiliar_Erro_Silo", PT := "DB_Geral".Time_TempoErro);
   IF "IEC_Timer_0_DB_TON_TempoErro".Q THEN #Falha_TimeOut_Desabastecimento := TRUE; END_IF;
END_REGION

REGION Network 11: Reset - Falhas
   RUNG wire#powerrail
      Contact( #iReset )
      wire#w1
      Contact( #Falha_TimeOut_Desabastecimento )
      R_Coil( #Falha_TimeOut_Desabastecimento )
   END_RUNG
   RUNG wire#w1
      Contact( #Falha_SensoresNivel )
      R_Coil( #Falha_SensoresNivel )
   END_RUNG
   // the same network as SCL:
   IF #iReset AND #Falha_TimeOut_Desabastecimento THEN #Falha_TimeOut_Desabastecimento := FALSE; END_IF;
   IF #iReset AND #Falha_SensoresNivel THEN #Falha_SensoresNivel := FALSE; END_IF;
END_REGION
END_FUNCTION

FUNCTION "FC_Silo_Principal" : Void   // FC6, LAD
{ S7_Optimized_Access := 'TRUE' }
VERSION : 0.1
   VAR_INPUT
      iAutomatico : Bool;
      iManual : Bool;
      iEmg : Bool;
      iReset : Bool;
      iBtnAbasteceSilo : Bool;
      iCmdAbasteceSilo : Bool;
      iSensorMaximo : Bool;
      iSensorMinimo : Bool;
   END_VAR
   VAR_OUTPUT
      oAbasteceSilo : Bool;
   END_VAR
   VAR_IN_OUT
      Falha_SensoresNivel : Bool;
      "Status Silo - Minimo" : Bool;
      "Status Silo - Maximo" : Bool;
      "Status Silo - Desabastecido" : Bool;
   END_VAR
BEGIN

REGION Network 1
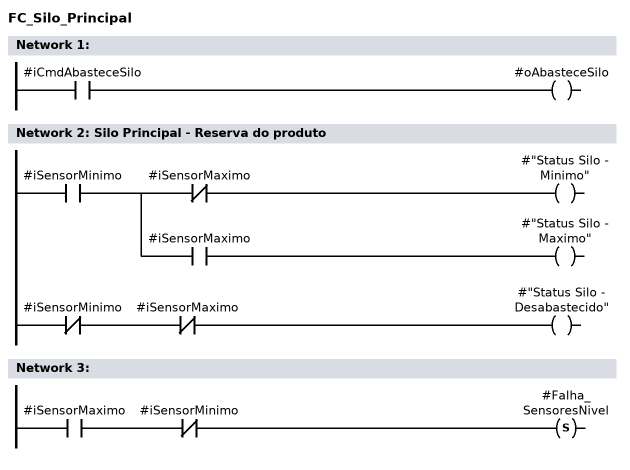
   RUNG wire#powerrail
      Contact( #iCmdAbasteceSilo )
      Coil( #oAbasteceSilo )
   END_RUNG
   // the same network as SCL:
   #oAbasteceSilo := #iCmdAbasteceSilo;
END_REGION

REGION Network 2: Silo Principal - Reserva do produto
   RUNG wire#powerrail
      Contact( #iSensorMinimo )
      wire#w1
      I_Contact( #iSensorMaximo )
      Coil( #"Status Silo - Minimo" )
   END_RUNG
   RUNG wire#w1
      Contact( #iSensorMaximo )
      Coil( #"Status Silo - Maximo" )
   END_RUNG
   RUNG wire#powerrail
      I_Contact( #iSensorMinimo )
      I_Contact( #iSensorMaximo )
      Coil( #"Status Silo - Desabastecido" )
   END_RUNG
   // the same network as SCL:
   #"Status Silo - Minimo" := #iSensorMinimo AND NOT #iSensorMaximo;
   #"Status Silo - Maximo" := #iSensorMinimo AND #iSensorMaximo;
   #"Status Silo - Desabastecido" := NOT #iSensorMinimo AND NOT #iSensorMaximo;
END_REGION

REGION Network 3
   RUNG wire#powerrail
      Contact( #iSensorMaximo )
      I_Contact( #iSensorMinimo )
      S_Coil( #Falha_SensoresNivel )
   END_RUNG
   // the same network as SCL:
   IF #iSensorMaximo AND NOT #iSensorMinimo THEN #Falha_SensoresNivel := TRUE; END_IF;
END_REGION
END_FUNCTION

ORGANIZATION_BLOCK "Main"   // OB1, LAD, ProgramCycle
TITLE = "Main Program Sweep (Cycle)"
{ S7_Optimized_Access := 'TRUE' }
VERSION : 0.1
   VAR_INPUT
      Initial_Call : Bool;   // Initial call of this OB
      Remanence : Bool;   // =True, if remanent data are available
   END_VAR
BEGIN
END_ORGANIZATION_BLOCK